TYPE "Ax_PB"
VERSION : 0.1
// Block: Ax_PB
   STRUCT
      Bwd_Minus : Bool;
      Fwd_Plus : Bool;
      MoveToPos : Bool;
   END_STRUCT;

END_TYPE
